(* CODESYS project 04_WagoAppDataLogger.ecp
   CompiledLibraryCompatibilityVersion: e!COCKPIT

Project tree, tasks and I/O mapping:
  PFC_Datalogger : 750-8212 PFC200 G2 2ETH RS, WAGO, order no. 0750-8212, version 5.16.3.16
    application Application
      libraries: ; WagoAppDatalogger, 1.0.2.0 (WAGO); VisuDialogs, * (System)
      task PLC_Task (cyclic, interval 50 ms, priority 15) calls PLC_PRG
      task VISU_TASK (cyclic, interval 100 ms, priority 15) calls VisuElems.Visu_Prg
      program PLC_PRG [ST]: actInit
      visualisation Visualization
    ProjectConfiguration
    ProjectConfigurationTxt
    Kbus : Kbus, WAGO, version 1.4.0.2
        unmapped channels: K-BUS diagnostics
    MODBUS
      MODBUS : MODBUS, WAGO, order no. n/a, version 1.1.1.16
    Serial
      COM1 : COM1, WAGO, version 0.0.0.19
    Common.PCI
    EtherNet/IP
      Ethernet : Ethernet, WAGO, version 35.16.0.0
  libraries: VisuSymbols, 3.5.10.0 (System); WagoVisuIcons, 1.1.0.3 (WAGO)
  text list GlobalTextList
  00000000-0000-0000-0000-000000000000|C:\Users\MarkusF\AppData\Local\Temp\85b4736708d94810a251f7ad5cab2671\Project.xml
  00000000-0000-0000-0000-000000000000|C:\Users\MarkusF\AppData\Local\Temp\13298d7665a846bfad5fcb3bd71d0184\ProjectCfg.txt
*)

// PFC_Datalogger/Application/PLC_PRG
PROGRAM PLC_PRG
VAR
	fbMyDataLogger:		WagoAppDatalogger.FbDatalogger;
	xEvent, xReady:		BOOL;
	xFirstCycle,
	xActivate:			BOOL := TRUE;
	aValues:			ARRAY [1..MAX_CHANNELS] OF REAL;
	sStatus:			STRING;
	Settings:			typConfigDatalogger;
	i:					INT;
	j, rSineL1, rSineL2, rSineL3, rTemperature: REAL;
	iTemp01Raw:			INT := 529;		// ==> 52.9 °C
END_VAR

// process the initialisation one time at the beginning
actInit();

// increment a real number veeery slowly
j := j + 0.002;
// create a three phase system with a peak value of 50.0,
// this is higher than some limits :-))
rSineL1			:= 50.0 * SIN(j);
rSineL2			:= 50.0 * SIN(j + 2.094395102393);
rSineL3			:= 50.0 * SIN(j + 4.188790204786);
// create some variation of the temperature
rTemperature	:= TO_REAL(iTemp01Raw) / 10.0 + 5* SIN(j);

// transfer the three sines and a temperature to the array
aValues[1]	:= rSineL1;
aValues[2]	:= rSineL2;
aValues[3]	:= rSineL3;
aValues[5]	:= rTemperature;

// run the datalogger
fbMyDataLogger(
	xActivate	:= xActivate,
	aValues		:= aValues,
	xEvent		:= xEvent,
	typConfigParameters := Settings,
	oStatus		=> ,
	sStatus		=> sStatus,
	xReady		=> xReady);

ACTION actInit:
IF xFirstCycle THEN
//	all comments taken from the help file, see WagoAppDatalogger.chm
(*	bDatalogger_type indicates which csv format should be used. There are 3 available formats:
	1) Standard Wago datalogger format
	2) Econ format
	3) Dataplotter format: Specific for the Dataplotter Web application. Please set MAX_CHANNELS
	   in ParameterList to 80. The dataplotter webapplication can only display up to 80 channels *)
	Settings.bDatalogger_type		:= 3;
//	automatically append current date to filename (new file each day!)
	Settings.xAppendDate			:= FALSE;
//	triggers the cyclic logging to the csv file
	Settings.xCyclicLogging			:= FALSE;
(*	bInterval defines the desired logging cycle unit:
	1) hours
	2) minutes
	3) seconds (default value) *)
	Settings.bInterval				:= 3;
	Settings.sFilename				:= 'logfile.csv';
//	this path must already exist on the sd card
	Settings.sPath					:= '/media/sd/CSV_Files/';
(*	decimal separator for values in csv file, default value is comma ','
	for the dataplotter-format, this parameter will be ignored. A full-stop '.' will always be used *)
	Settings.sDecimalSeparator		:=',';
(*	column separator in csv file, default-value is comma ';'
	for the dataplotter-format, this parameter will be ignored. A comma ',' will always be used *)
	Settings.sColumnSeparator		:=';';
//	desired logging factor factor (default value = 1, max value = 65535)
	Settings.uiIntervalFactor		:= 1;

(*	will be executed only once after start of program to enable editable channel variables
	set all channels to false *)
	FOR i := 1 TO 80 DO
		Settings.atypChannelConfig[i].xChannelExists := FALSE;
	END_FOR

	Settings.atypChannelConfig[1].xChannelExists	:= TRUE;
	Settings.atypChannelConfig[1].bDecimalPlaces	:= 2;			// number of digits after the decimal-point, if not specified: default-value = 2
	Settings.atypChannelConfig[1].xLogAlarm			:= TRUE;		// shows alarm column of sine-function in file (for standard datalogger)
	Settings.atypChannelConfig[1].sChannelName		:= 'Sine Curve L1';
	Settings.atypChannelConfig[1].sUnit				:= 'V';
	Settings.atypChannelConfig[1].rAlarmLowerLimit	:= -40;
	Settings.atypChannelConfig[1].rAlarmUpperLimit	:= 40;

	Settings.atypChannelConfig[2].xChannelExists	:= TRUE;
	Settings.atypChannelConfig[2].bDecimalPlaces	:= 2;
	Settings.atypChannelConfig[2].xLogAlarm			:= TRUE;
	Settings.atypChannelConfig[2].sChannelName		:= 'Sine Curve L2';
	Settings.atypChannelConfig[2].sUnit				:= 'V';
	Settings.atypChannelConfig[2].rAlarmLowerLimit	:= -40;
	Settings.atypChannelConfig[2].rAlarmUpperLimit	:= 48;

	Settings.atypChannelConfig[3].xChannelExists	:= TRUE;
	Settings.atypChannelConfig[3].bDecimalPlaces	:= 2;
	Settings.atypChannelConfig[3].xLogAlarm			:= TRUE;
	Settings.atypChannelConfig[3].sChannelName		:= 'Sine Curve L3';
	Settings.atypChannelConfig[3].sUnit				:= 'V';
	Settings.atypChannelConfig[3].rAlarmLowerLimit	:= -40;
	Settings.atypChannelConfig[3].rAlarmUpperLimit	:= 48;

	Settings.atypChannelConfig[5].xChannelExists	:= TRUE;
	Settings.atypChannelConfig[5].bDecimalPlaces	:= 2;
	Settings.atypChannelConfig[5].xLogAlarm			:= TRUE;
	Settings.atypChannelConfig[5].sChannelName		:= 'Temperature';
	Settings.atypChannelConfig[5].sUnit				:= '°C';
	Settings.atypChannelConfig[5].rAlarmLowerLimit	:= -0;
	Settings.atypChannelConfig[5].rAlarmUpperLimit	:= 40;

	xFirstCycle := FALSE;		// prevents another call of initialization

END_IF

// entries outside of IF-THEN construct will be executed in each cycle of the PLC
END_ACTION

END_PROGRAM

// PFC_Datalogger/Application/Visualization
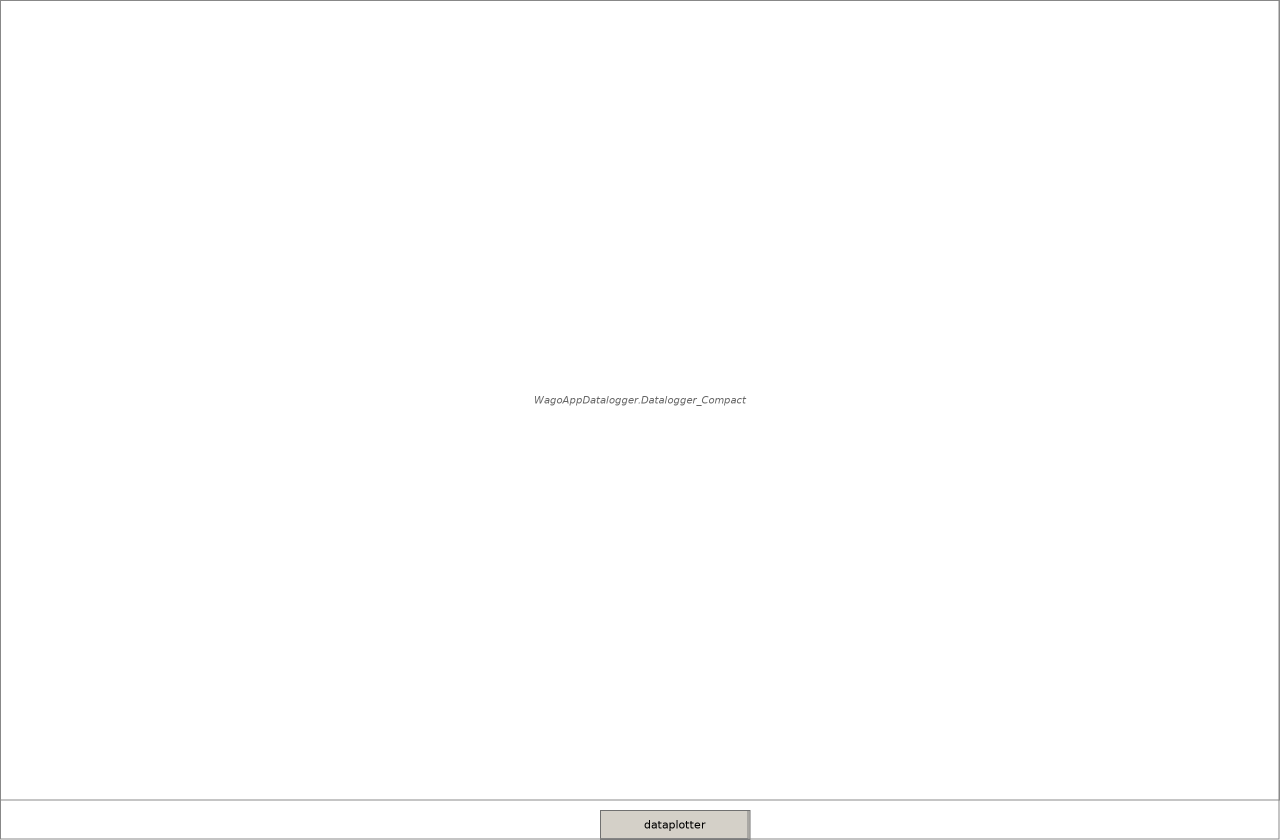
VISUALIZATION Visualization  // 1280x840
    Frame (0,0 1280x800)
        shows WagoAppDatalogger.Datalogger_Compact(oDatalogger := PLC_PRG.fbMyDataLogger)
        shows WagoAppDatalogger.Channels(oDatalogger := PLC_PRG.myDataLogger)
        shows WagoAppDatalogger.MessageBar(oDatalogger := PLC_PRG.myDataLogger)
        shows WagoAppDatalogger.RibbonBarFileSettings(oDatalogger := PLC_PRG.myDataLogger)
        shows WagoAppDatalogger.StatusBar(oDatalogger := PLC_PRG.myDataLogger)
    Button (600,810 150x30), "dataplotter"
        OnMouseUp:  ExecuteCommand=ExecuteCommand=[Command=NavigateURL, Value='http://192.168.1.123/dataplotter/dataplotter.html']
END_VISUALIZATION
